ABB RobotStudio station: apilar_yogur.rspag

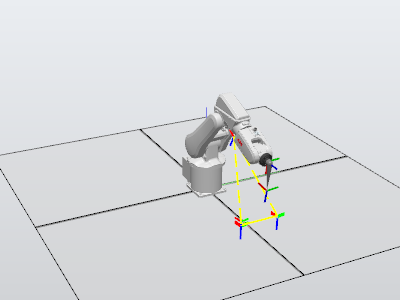
--- station ---
Station Project3 (saved by RobotStudio 25.3.11371.0)
Controller IRB120_3_58
  mechanical unit ROB_1: IRB120_3_58__01, 6 joints, base frame (0, 0, 0) mm
Layout (positions relative to the parent item):
  - IRB120_3_58__01 [mechanism, from %ABB.RobotStudio.Models.IRB120%\IRB120_3_58_G_01.rslib] at (0, 0, 0) mm; joint values [0.1187, 0.7429, -0.21, -0.0058, -0.3449, 0.0138] (rad or m)
  - ventosa [mechanism] at (545.17, 65.15, 382.25) mm, rotated rx 177.38 ry 79.21 rz -175.75 deg
      TCP ventosa at (160, 0, 30) mm, rotated rx 0 ry 90 rz 0 deg
      links: Dummy
  - SmartComponent_1 [smart component]
      signals: DI coger, DO cogido, DI poner_yogur
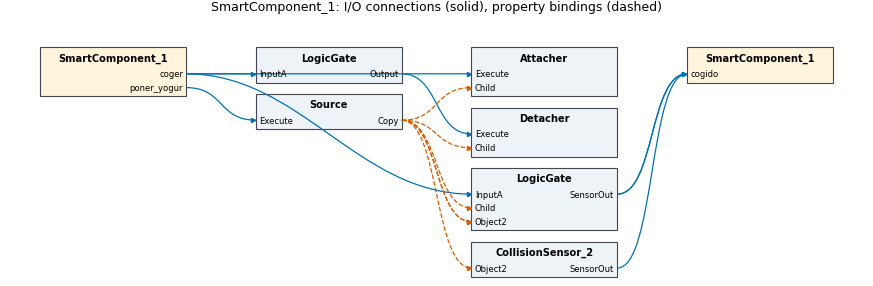
      connections:
        SmartComponent_1.coger -> LogicGate.InputA
        CollisionSensor.SensorOut -> SmartComponent_1.cogido
        SmartComponent_1.poner_yogur -> Source.Execute
        SmartComponent_1.coger -> Attacher.Execute
        LogicGate.Output -> Detacher.Execute
        SmartComponent_1.coger -> LogicGate.InputA
        CollisionSensor.SensorOut -> SmartComponent_1.cogido
        CollisionSensor_2.SensorOut -> SmartComponent_1.cogido
        Source.Copy => Attacher.Child
        Source.Copy => CollisionSensor.Object2
        Source.Copy => Attacher.Child
        Source.Copy => Detacher.Child
        Source.Copy => CollisionSensor.Object2
        Source.Copy => CollisionSensor_2.Object2
    - Yogur [part] at (590, 107, 0) mm, size 55 x 54.6 x 66 mm
    - Source [smart component, from Components\Source.rslib]
        properties: Source=Yogur; Copy=(none); Parent=(none); Position=[0.59 0.107 0]; Orientation=[0 0 0]; Transient=true; PhysicsBehavior=3
    - Attacher [smart component, from Components\Attacher.rslib]
        properties: Parent=ventosa; Flange=0; Child=(none); Mount=false; Offset=[0 0 0]; Orientation=[0 0 0]
    - Detacher [smart component, from Components\Detacher.rslib]
        properties: Child=(none); KeepPosition=true
    - LogicGate [smart component, from Components\LogicGate.rslib]
        properties: Operator=NOT; Delay=0
    - CollisionSensor_2 [smart component, from Components\CollisionSensor.rslib]
        properties: Object1=ventosa; Object2=(none); NearMiss=0.066; Part1=(none); Part2=(none); CollisionType=0
      - _sensorPart_ [part]
Attachment: ventosa is attached to IRB120_3_58__01 / Link6
Station signals: DI SacarYogur
Station logic (signal -> signal, property => property):
  IRB120_3_58.Do_0 -> SmartComponent_1.coger
  SmartComponent_1.cogido -> IRB120_3_58.Di_0

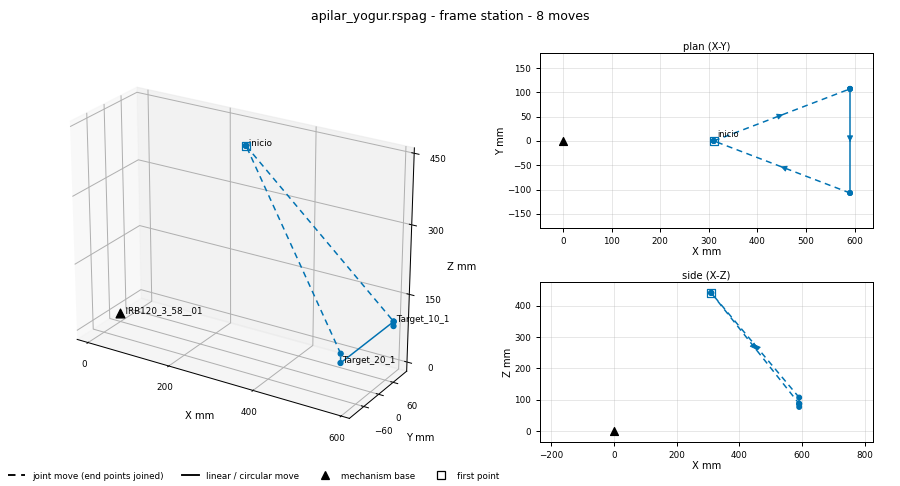
[picture p0: tool path of apilar_yogur.rspag in frame station, 8 of 8 moves have a stored position in this frame; points joined in program order, loops and branches not executed]
--- Controller Data/IRB120_3_58/RAPID/TASK1/PROGMOD/CalibData.mod ---
MODULE CalibData
    PERS tooldata ventosa:=[TRUE,[[160,0,30],[0.707106781,0,0.707106781,0]],[1,[0,0,1],[1,0,0,0],0,0,0]];
    TASK PERS wobjdata Workobject_1:=[FALSE,TRUE,"",[[0,0,0],[1,0,0,0]],[[0,0,0],[1,0,0,0]]];
ENDMODULE

--- Controller Data/IRB120_3_58/RAPID/TASK1/PROGMOD/Module1.mod ---
MODULE Module1
    CONST robtarget inicio:=[[310.334591186,0,440.435935394],[0.258819045,0,-0.965925826,0],[0,0,0,0],[9E+09,9E+09,9E+09,9E+09,9E+09,9E+09]];
    CONST robtarget Target_10:=[[590.589058249,107.133669034,77.210444148],[0.015424305,0.090036277,-0.995802425,-0.005752415],[0,-1,0,1],[9E+09,9E+09,9E+09,9E+09,9E+09,9E+09]];
    CONST robtarget Target_10_1:=[[590.589058249,107.133669034,87.210444148],[0.015424305,0.090036277,-0.995802425,-0.005752415],[0,-1,0,1],[9E+09,9E+09,9E+09,9E+09,9E+09,9E+09]];
    CONST robtarget Target_20_1:=[[590.589058249,-107.133669034,87.210444148],[0.015424305,0.090036277,-0.995802425,-0.005752415],[0,-1,0,1],[9E+09,9E+09,9E+09,9E+09,9E+09,9E+09]];
     CONST robtarget Target_20_2:=[[590.589058249,-107.133669034,107.210444148],[0.015424305,0.090036277,-0.995802425,-0.005752415],[0,-1,0,1],[9E+09,9E+09,9E+09,9E+09,9E+09,9E+09]];
    CONST robtarget Target_20:=[[590.589058249,-107.133669034,77.210444148],[0.015424305,0.090036277,-0.995802425,-0.005752415],[0,-1,0,1],[9E+09,9E+09,9E+09,9E+09,9E+09,9E+09]];
    PROC Path_10()
        MoveJ inicio,v100,z100,ventosa\WObj:=Workobject_1;

        MoveJ Target_10_1,v100,z0,ventosa\WObj:=Workobject_1;
       WaitTime 1;
        IF Di_0=1 THEN
             MoveJDO Target_10,v100,z0,ventosa\WObj:=Workobject_1, Do_0,1;
        MoveJ Target_10_1,v100,z0,ventosa\WObj:=Workobject_1;
    !Set Do_0;
        MoveL Target_20_1,v100,z0,ventosa\WObj:=Workobject_1;


          MoveJDO Target_20_2,v500,z0,ventosa\WObj:=Workobject_1, Do_0,0;
        MoveJ inicio,v500,z100,ventosa\WObj:=Workobject_1;
        ELSE
          Reset Do_0;
          MoveJ inicio,v500,z100,ventosa\WObj:=Workobject_1;
        ENDIF
    ENDPROC
    PROC main()
        Path_10;
    ENDPROC
ENDMODULE

--- Controller Data/IRB120_3_58/SYSPAR/EIO.cfg ---
EIO:CFG_1.0:6:1::
#
INDUSTRIAL_NETWORK:

      -Name "DeviceNet" -Label "DeviceNet Master/Slave Network" -Address "2"
#
DEVICENET_DEVICE:

      -Name "d652" -VendorName "ABB Robotics" -ProductName "24 VDC I/O Device"\
      -Label "DSQC 652 24 VDC I/O Device" -Address 10 -ProductCode 26\
      -DeviceType 7 -ConnectionType "COS" -OutputSize 2 -InputSize 2
#
DEVICENET_INTERNAL_DEVICE:

      -Name "DN_Internal_Device" -VendorName "ABB Robotics"\
      -ProductName "DeviceNet Internal Slave Device"
#
EIO_SIGNAL:

      -Name "Di_0" -SignalType "DI" -Device "d652" -DeviceMap "0" -Access "All"

      -Name "Do_0" -SignalType "DO" -Device "d652" -DeviceMap "0" -Access "All"
